// Mitsubishi GX Works2 project: EX2 (1) (1)   PLC: FX3G

// global labels: Global1
VAR_GLOBAL
  RM_Petel_Input AT D1100 : REAL;
  RG_Petel_Input AT D1100 : REAL;
  RG_Petel_Count AT D1200 : REAL;
  RG_Lemon_Input AT D1105 : REAL;
  RG_Lemon_Count AT D1205 : REAL;
  RG_Bear_Input AT D1110 : REAL;
  RG_Bear_Count AT D1215 : REAL;
  RG_Stables_Input AT D1120 : REAL;
  RG_Stables_Count AT D1220 : REAL;
END_VAR
VAR_GLOBAL CONSTANT
  Min_Petel_Amout : REAL := 385;
END_VAR
VAR_GLOBAL
  M2_Have_Petel AT M2 : BOOL;
END_VAR
VAR_GLOBAL CONSTANT
  Min_Petel_Amount : REAL := 105;
END_VAR
VAR_GLOBAL
  M3_Have_Lemon AT M3 : BOOL;
END_VAR
VAR_GLOBAL CONSTANT
  Min_Lemon_Amount : REAL := 665;
  Min_Bear_Amount : REAL := 70;
END_VAR
VAR_GLOBAL
  M4_Have_Bear AT M4 : BOOL;
END_VAR
VAR_GLOBAL CONSTANT
  Min_Stables_Amount : REAL := 210;
END_VAR
VAR_GLOBAL
  M5_Have_Stables AT M5 : BOOL;
  RG_Sample_Type_Value AT D1500 : REAL;
END_VAR
VAR_GLOBAL CONSTANT
  Con400 : INT := K400;
  Cons400 : REAL := 400;
END_VAR
VAR_GLOBAL
  M9_select_type AT M9 : BOOL;
END_VAR
VAR_GLOBAL CONSTANT
  Cons5 : REAL := 5;
END_VAR
VAR_GLOBAL
  TS5_end_making AT TS5 : BOOL;
  M91_regular AT M91 : BOOL;
END_VAR
VAR_GLOBAL CONSTANT
  Cons6 : REAL := 6;
  Cons10 : INT := 10;
END_VAR
VAR_GLOBAL
  TS6_end_making AT TS6 : BOOL;
  M92_pinok AT M92 : BOOL;
END_VAR
VAR_GLOBAL CONSTANT
  Petel_Amount : REAL := 280;
END_VAR
VAR_GLOBAL
  RG_Petel_Making AT D1400 : REAL;
END_VAR
VAR_GLOBAL CONSTANT
  Lemon_Amount_Petel : REAL := 35;
  Lemon_Amount_Lemon : REAL := 420;
END_VAR
VAR_GLOBAL
  RG_Lemon_Making AT D1410 : REAL;
END_VAR
VAR_GLOBAL CONSTANT
  Stables_Amount_Petel : REAL := 35;
  Steables_Amount_Lemon : REAL := 70;
  Petel_Amount_pinok : REAL := 385;
  Lemon_Amount_Petel_Pinok : REAL := 105;
  Lemon_Amount_Lemon_Pinok : REAL := 560;
  Stables_Amount_Petel_Pinok : REAL := 70;
  Steables_Amount_Lemon_Pinok : REAL := 140;
  Lemon_Amount_total : REAL := 455;
  Stables_Amount_total : REAL := 105;
  Lemon_Amount_total_pinok : REAL := 665;
  Stables_Amount_total_pinok : REAL := 210;
  Count5 : REAL := 5;
  Cons50 : WORD := 50;
  Cons0 : REAL;
END_VAR
VAR_GLOBAL
  RG_type_analog_value AT D1610 : REAL;
  X6Test AT X006 : BOOL;
  RG_Petel_Cooling AT D1404 : REAL;
  RG_Lemon_Cooling AT D1414 : REAL;
  TC7_cooling AT TC7 : BOOL;
END_VAR
VAR_GLOBAL CONSTANT
  Cons80 : WORD := 80;
END_VAR
VAR_GLOBAL
  M11_cooling AT M11 : BOOL;
  TS7_end_cooling AT TS7 : BOOL;
  Y4_TEST AT Y004 : BOOL;
END_VAR
VAR_GLOBAL CONSTANT
  Regular_Bear : REAL := 28;
END_VAR
VAR_GLOBAL
  RG_Mix_Regular AT D1450 : REAL;
END_VAR
VAR_GLOBAL CONSTANT
  Pinok_Bear : REAL := 70;
END_VAR
VAR_GLOBAL
  RG_Mix_Pinok AT D1460 : REAL;
  TC8_Mixing_Regular AT TC8 : BOOL;
END_VAR
VAR_GLOBAL CONSTANT
  Cons30 : WORD := 30;
END_VAR
VAR_GLOBAL
  TC9_Mixing_Pinok AT TC9 : BOOL;
  M10_Mixing AT M10 : BOOL;
  TS8_End_Mixing_Regual AT TS8 : BOOL;
  M0_Mix_Blinking AT M0 : BOOL;
  TS0_Output_Timer AT TS0 : BOOL;
  M20_Mix_Blinking_Help1 AT M20 : BOOL;
  TC0_Blinking1_Timer AT TC0 : BOOL;
  TC1_Blinking2_Timer AT TC1 : BOOL;
  TS1_Output_Timer2 AT TS1 : BOOL;
  M21_Mix_Blinking_Help2 AT M21 : BOOL;
  TS9_End_Mixing_Pinok AT TS9 : BOOL;
END_VAR
VAR_GLOBAL CONSTANT
  Const10 : REAL := 10;
END_VAR
VAR_GLOBAL
  X4_Packing AT X004 : BOOL;
  X0_packing_1_ice_cream AT X000 : BOOL;
  Y4_Work_ON_packing AT Y004 : BOOL;
END_VAR
VAR_GLOBAL CONSTANT
  Cons7 : WORD := 7;
END_VAR
VAR_GLOBAL
  RG_Ice_Output AT D1600 : REAL;
  RG_Packed_Ice_Cream AT D1700 : REAL;
END_VAR
VAR_GLOBAL CONSTANT
  Con1 : REAL := 1;
  Cons40 : REAL := 40;
END_VAR
VAR_GLOBAL
  RG_Packed_Ice_Cream_float AT D1710 : REAL;
  Y7_Working_day AT Y007 : BOOL;
  X5_Emergency AT X005 : BOOL;
  M7_End_Of_Day AT M7 : BOOL;
  X7_Start_Day AT X007 : BOOL;
  X1_Sample_Type AT X001 : BOOL;
  Y0_making AT Y000 : BOOL;
  X2_Cooling AT X002 : BOOL;
  Y2_Cooling AT Y002 : BOOL;
  X3_Temp AT X003 : BOOL;
  TC5_making AT TC5 : BOOL;
  TC6_making AT TC6 : BOOL;
  M15_packing AT M15 : BOOL;
  Y5_Mixing AT Y005 : BOOL;
  Y6_Mixing AT Y006 : BOOL;
  CS1_Packing_Finish AT CS1 : BOOL;
  CC1_Packing AT CC1 : BOOL;
  M12_end_cooling AT M12 : BOOL;
  M16_End_Packing AT M16 : BOOL;
  M17_packing_help AT M17 : BOOL;
  RG_analog2_Output AT D8282 : INT;
  RG_Sample_Type AT D8280 : INT;
END_VAR

// task Task_01 (event TRUE, interval 0, priority 31): POU_01

PROGRAM POU_01
(* structured ladder/FBD written out as ST: instructions are called as NAME(EN, inputs, outputs); _pN, _eN, _tN stand for wires *)
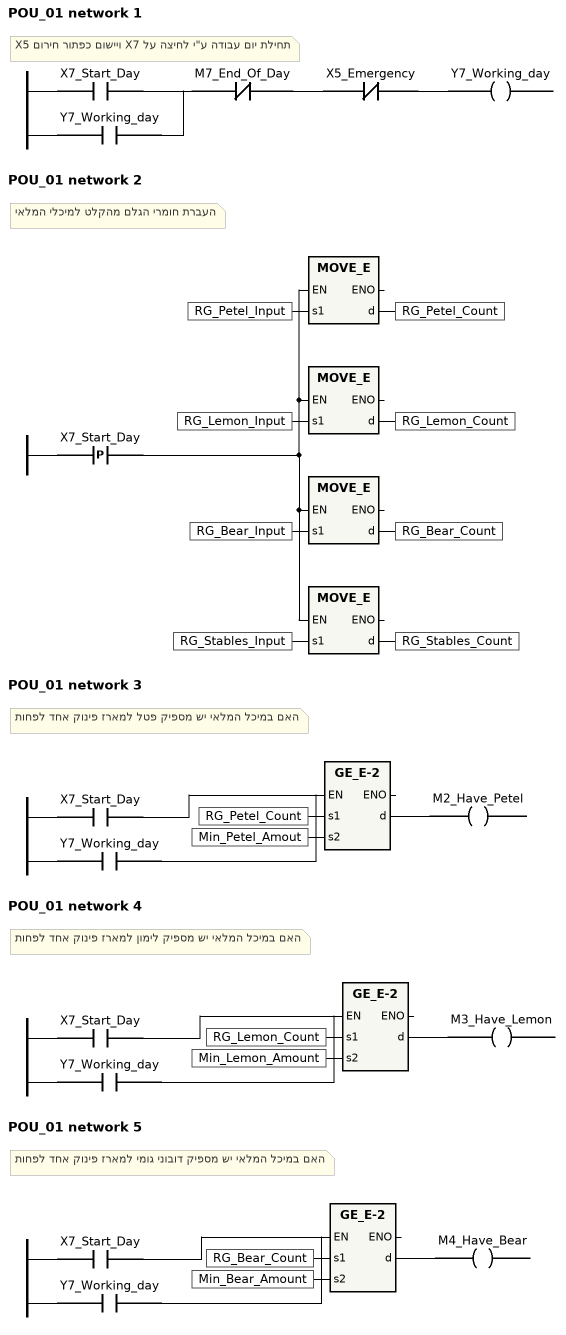
(* network 1 *)
(* תחילת יום עבודה ע"י לחיצה על X7 ויישום כפתור חירום X5 *)
Y7_Working_day := ((X7_Start_Day OR Y7_Working_day) AND NOT M7_End_Of_Day) AND NOT X5_Emergency;
(* network 2 *)
(* העברת חומרי הגלם מהקלט למיכלי המלאי *)
_p1 := LDP(TRUE, X7_Start_Day);
MOVE_E(_p1, RG_Petel_Input, RG_Petel_Count);
MOVE_E(_p1, RG_Lemon_Input, RG_Lemon_Count);
MOVE_E(_p1, RG_Bear_Input, RG_Bear_Count);
MOVE_E(_p1, RG_Stables_Input, RG_Stables_Count);
(* network 3 *)
(* האם במיכל המלאי יש מספיק פטל למארז פינוק אחד לפחות *)
GE_E(X7_Start_Day OR Y7_Working_day, RG_Petel_Count, Min_Petel_Amout, _t1);
M2_Have_Petel := _t1;
(* network 4 *)
(* האם במיכל המלאי יש מספיק לימון למארז פינוק אחד לפחות *)
GE_E(X7_Start_Day OR Y7_Working_day, RG_Lemon_Count, Min_Lemon_Amount, _t1);
M3_Have_Lemon := _t1;
(* network 5 *)
(* האם במיכל המלאי יש מספיק דובוני גומי למארז פינוק אחד לפחות *)
GE_E(X7_Start_Day OR Y7_Working_day, RG_Bear_Count, Min_Bear_Amount, _t1);
M4_Have_Bear := _t1;
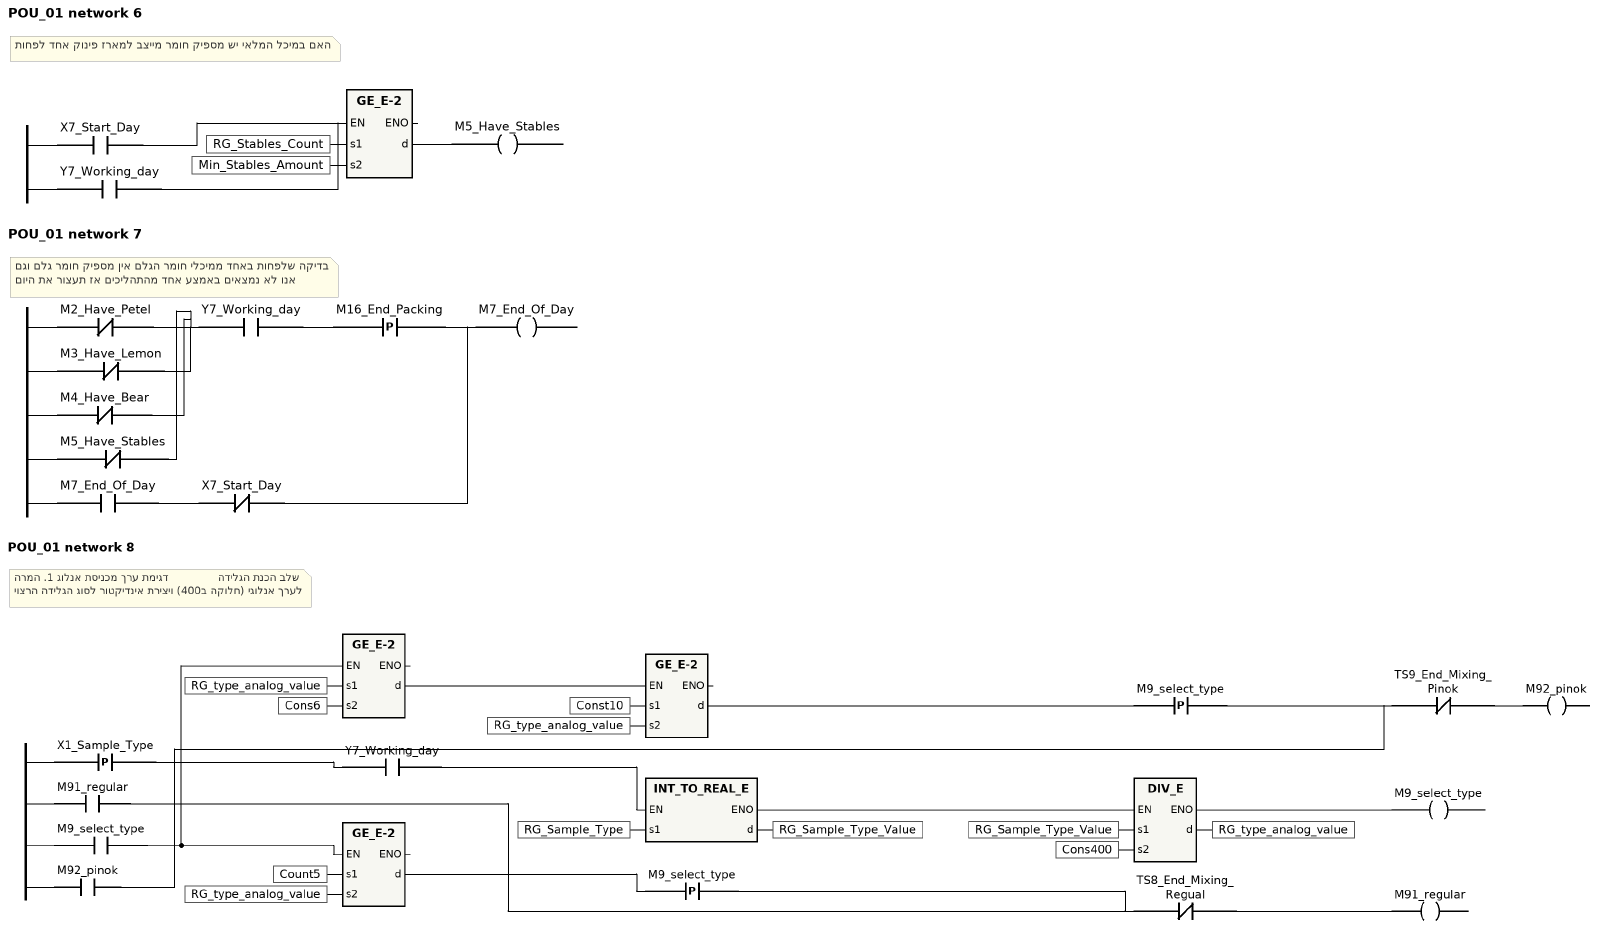
(* network 6 *)
(* האם במיכל המלאי יש מספיק חומר מייצב למארז פינוק אחד לפחות *)
GE_E(X7_Start_Day OR Y7_Working_day, RG_Stables_Count, Min_Stables_Amount, _t1);
M5_Have_Stables := _t1;
(* network 7 *)
(* בדיקה שלפחות באחד ממיכלי חומר הגלם אין מספיק חומר גלם וגם אנו לא נמצאים באמצע אחד מהתהליכים אז תעצור את היום *)
M7_End_Of_Day := ((((NOT M2_Have_Petel) OR (NOT M3_Have_Lemon) OR (NOT M4_Have_Bear) OR (NOT M5_Have_Stables)) AND Y7_Working_day) AND LDP(TRUE, M16_End_Packing)) OR (M7_End_Of_Day AND NOT X7_Start_Day);
(* network 8 *)
(* שלב הכנת הגלידה               דגימת ערך מכניסת אנלוג 1. המרה לערך אנלוגי (חלוקה ב400) ויצירת אינדיקטור לסוג הגלידה הרצוי *)
_e1 := INT_TO_REAL_E(LDP(TRUE, X1_Sample_Type) AND Y7_Working_day, RG_Sample_Type, RG_Sample_Type_Value);
_e2 := DIV_E(_e1, RG_Sample_Type_Value, Cons400, RG_type_analog_value);
M9_select_type := _e2;
GE_E(M9_select_type, Count5, RG_type_analog_value, _t3);
M91_regular := (M91_regular OR (_t3 AND LDP(TRUE, M9_select_type))) AND NOT TS8_End_Mixing_Regual;
GE_E(M9_select_type, RG_type_analog_value, Cons6, _t4);
GE_E(_t4, Const10, RG_type_analog_value, _t5);
M92_pinok := ((_t5 AND LDP(TRUE, M9_select_type)) OR M92_pinok) AND NOT TS9_End_Mixing_Pinok;
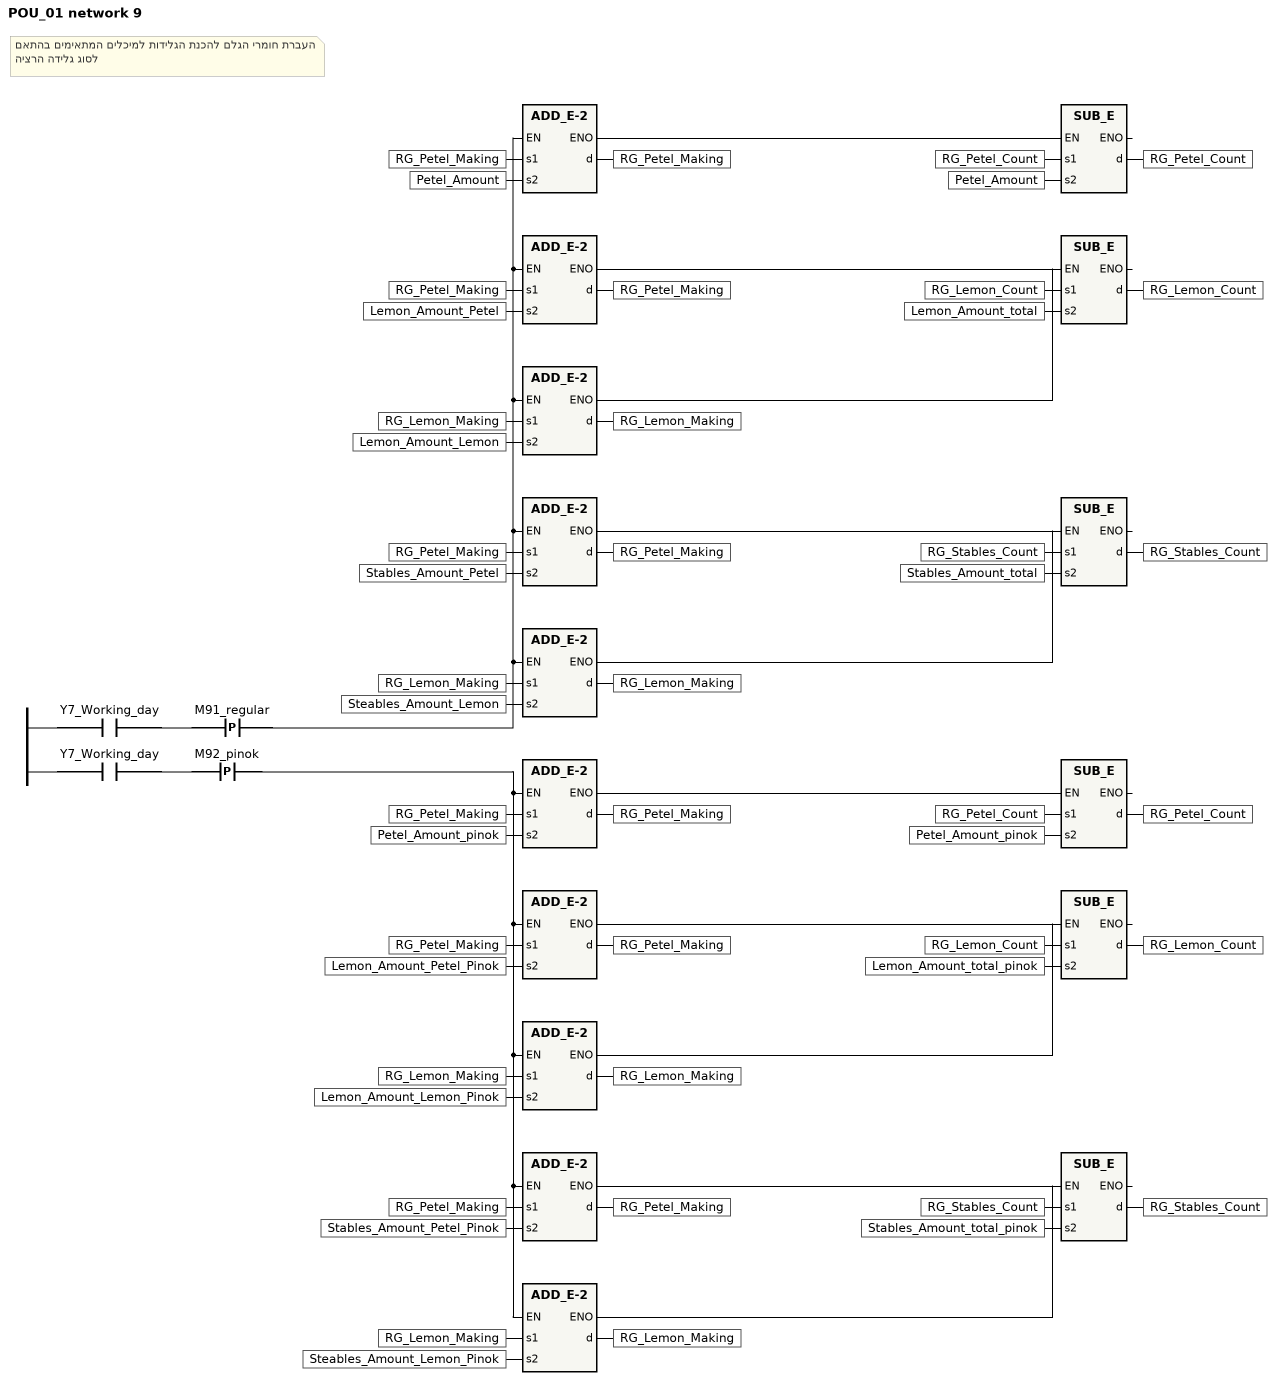
(* network 9 *)
(* העברת חומרי הגלם להכנת הגלידות למיכלים המתאימים בהתאם לסוג גלידה הרציה *)
_p1 := Y7_Working_day AND LDP(TRUE, M91_regular);
_e2 := ADD_E(_p1, RG_Petel_Making, Petel_Amount, RG_Petel_Making);
SUB_E(_e2, RG_Petel_Count, Petel_Amount, RG_Petel_Count);
_e3 := ADD_E(_p1, RG_Petel_Making, Lemon_Amount_Petel, RG_Petel_Making);
_e4 := ADD_E(_p1, RG_Lemon_Making, Lemon_Amount_Lemon, RG_Lemon_Making);
SUB_E(_e3 OR _e4, RG_Lemon_Count, Lemon_Amount_total, RG_Lemon_Count);
_e5 := ADD_E(_p1, RG_Petel_Making, Stables_Amount_Petel, RG_Petel_Making);
_e6 := ADD_E(_p1, RG_Lemon_Making, Steables_Amount_Lemon, RG_Lemon_Making);
SUB_E(_e5 OR _e6, RG_Stables_Count, Stables_Amount_total, RG_Stables_Count);
_p7 := Y7_Working_day AND LDP(TRUE, M92_pinok);
_e8 := ADD_E(_p7, RG_Petel_Making, Petel_Amount_pinok, RG_Petel_Making);
SUB_E(_e8, RG_Petel_Count, Petel_Amount_pinok, RG_Petel_Count);
_e9 := ADD_E(_p7, RG_Petel_Making, Lemon_Amount_Petel_Pinok, RG_Petel_Making);
_e10 := ADD_E(_p7, RG_Lemon_Making, Lemon_Amount_Lemon_Pinok, RG_Lemon_Making);
SUB_E(_e9 OR _e10, RG_Lemon_Count, Lemon_Amount_total_pinok, RG_Lemon_Count);
_e11 := ADD_E(_p7, RG_Petel_Making, Stables_Amount_Petel_Pinok, RG_Petel_Making);
_e12 := ADD_E(_p7, RG_Lemon_Making, Steables_Amount_Lemon_Pinok, RG_Lemon_Making);
SUB_E(_e11 OR _e12, RG_Stables_Count, Stables_Amount_total_pinok, RG_Stables_Count);
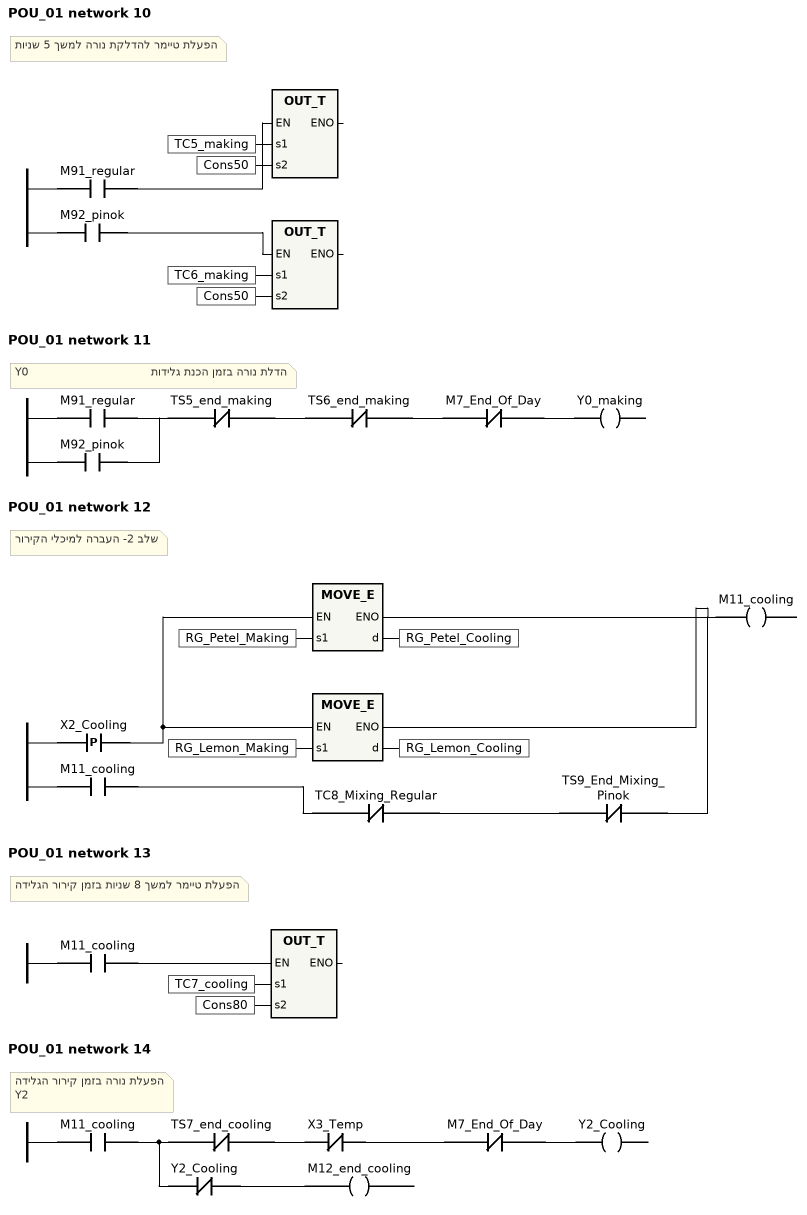
(* network 10 *)
(* הפעלת טיימר להדלקת נורה למשך 5 שניות *)
OUT_T(M91_regular, TC5_making, Cons50);
OUT_T(M92_pinok, TC6_making, Cons50);
(* network 11 *)
(* הדלת נורה בזמן הכנת גלידות                                   Y0 *)
Y0_making := (((M91_regular OR M92_pinok) AND NOT TS5_end_making) AND NOT TS6_end_making) AND NOT M7_End_Of_Day;
(* network 12 *)
(* שלב 2- העברה למיכלי הקירור *)
_p1 := LDP(TRUE, X2_Cooling);
_e2 := MOVE_E(_p1, RG_Petel_Making, RG_Petel_Cooling);
_e3 := MOVE_E(_p1, RG_Lemon_Making, RG_Lemon_Cooling);
M11_cooling := _e2 OR _e3 OR (M11_cooling AND NOT TC8_Mixing_Regular AND NOT TS9_End_Mixing_Pinok);
(* network 13 *)
(* הפעלת טיימר למשך 8 שניות בזמן קירור הגלידה *)
OUT_T(M11_cooling, TC7_cooling, Cons80);
(* network 14 *)
(* הפעלת נורה בזמן קירור הגלידה  / Y2 *)
Y2_Cooling := M11_cooling AND NOT TS7_end_cooling AND NOT X3_Temp AND NOT M7_End_Of_Day;
M12_end_cooling := M11_cooling AND NOT Y2_Cooling;
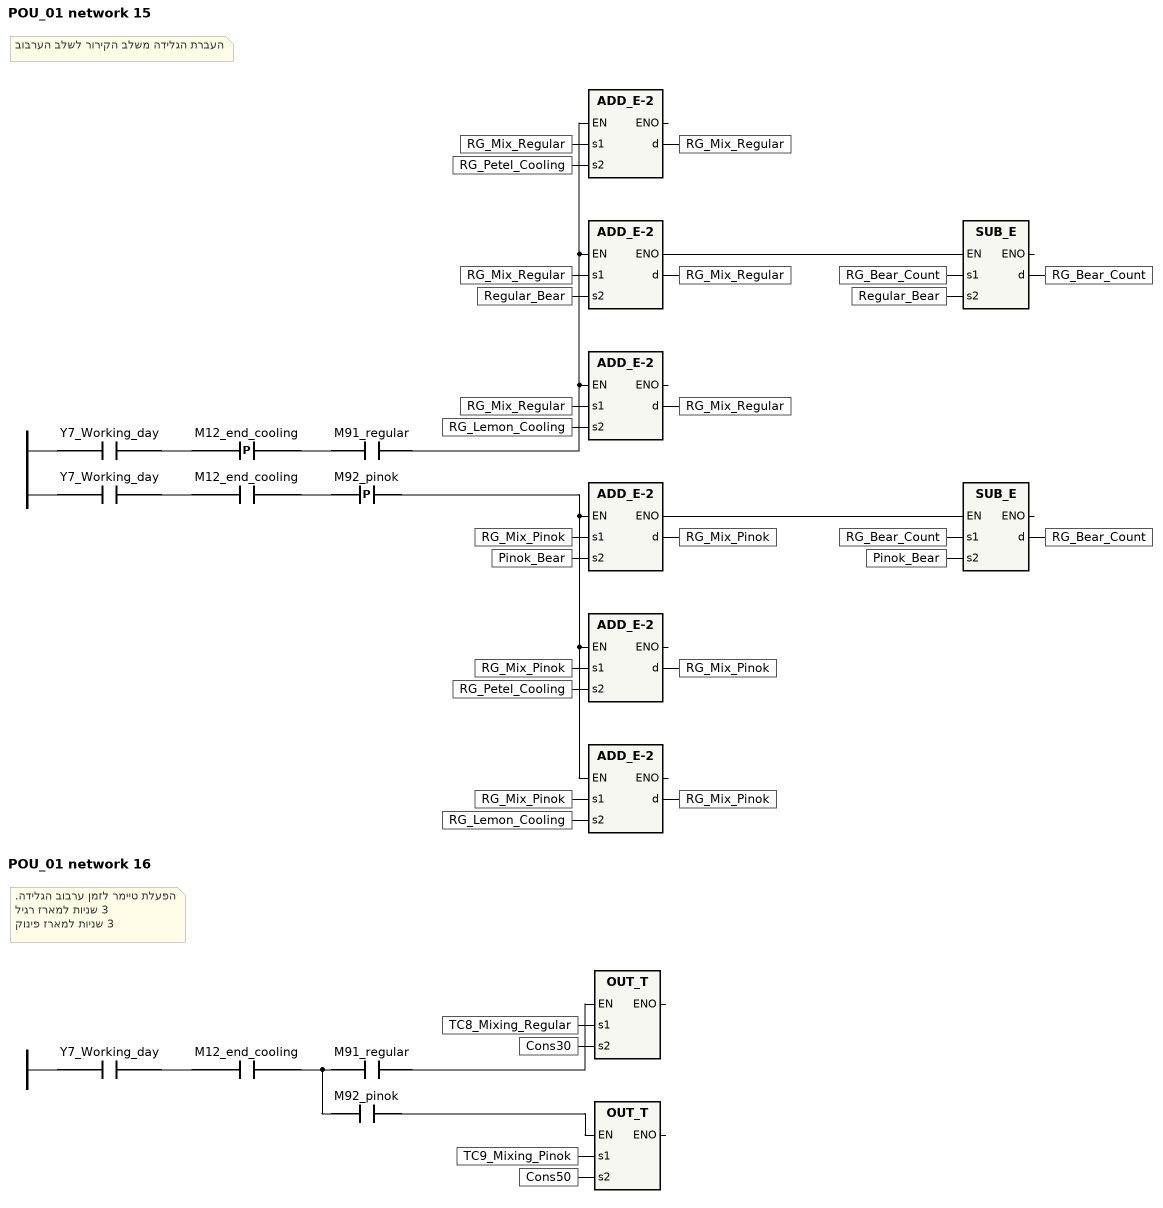
(* network 15 *)
(* העברת הגלידה משלב הקירור לשלב הערבוב *)
_p1 := Y7_Working_day AND LDP(TRUE, M12_end_cooling) AND M91_regular;
ADD_E(_p1, RG_Mix_Regular, RG_Petel_Cooling, RG_Mix_Regular);
ADD_E(_p1, RG_Mix_Regular, RG_Lemon_Cooling, RG_Mix_Regular);
_e2 := ADD_E(_p1, RG_Mix_Regular, Regular_Bear, RG_Mix_Regular);
SUB_E(_e2, RG_Bear_Count, Regular_Bear, RG_Bear_Count);
_p3 := Y7_Working_day AND M12_end_cooling AND LDP(TRUE, M92_pinok);
ADD_E(_p3, RG_Mix_Pinok, RG_Petel_Cooling, RG_Mix_Pinok);
ADD_E(_p3, RG_Mix_Pinok, RG_Lemon_Cooling, RG_Mix_Pinok);
_e4 := ADD_E(_p3, RG_Mix_Pinok, Pinok_Bear, RG_Mix_Pinok);
SUB_E(_e4, RG_Bear_Count, Pinok_Bear, RG_Bear_Count);
(* network 16 *)
(* הפעלת טיימר לזמן ערבוב הגלידה. / 3 שניות למארז רגיל / 3 שניות למארז פינוק *)
_p1 := Y7_Working_day AND M12_end_cooling;
OUT_T(_p1 AND M91_regular, TC8_Mixing_Regular, Cons30);
OUT_T(_p1 AND M92_pinok, TC9_Mixing_Pinok, Cons50);
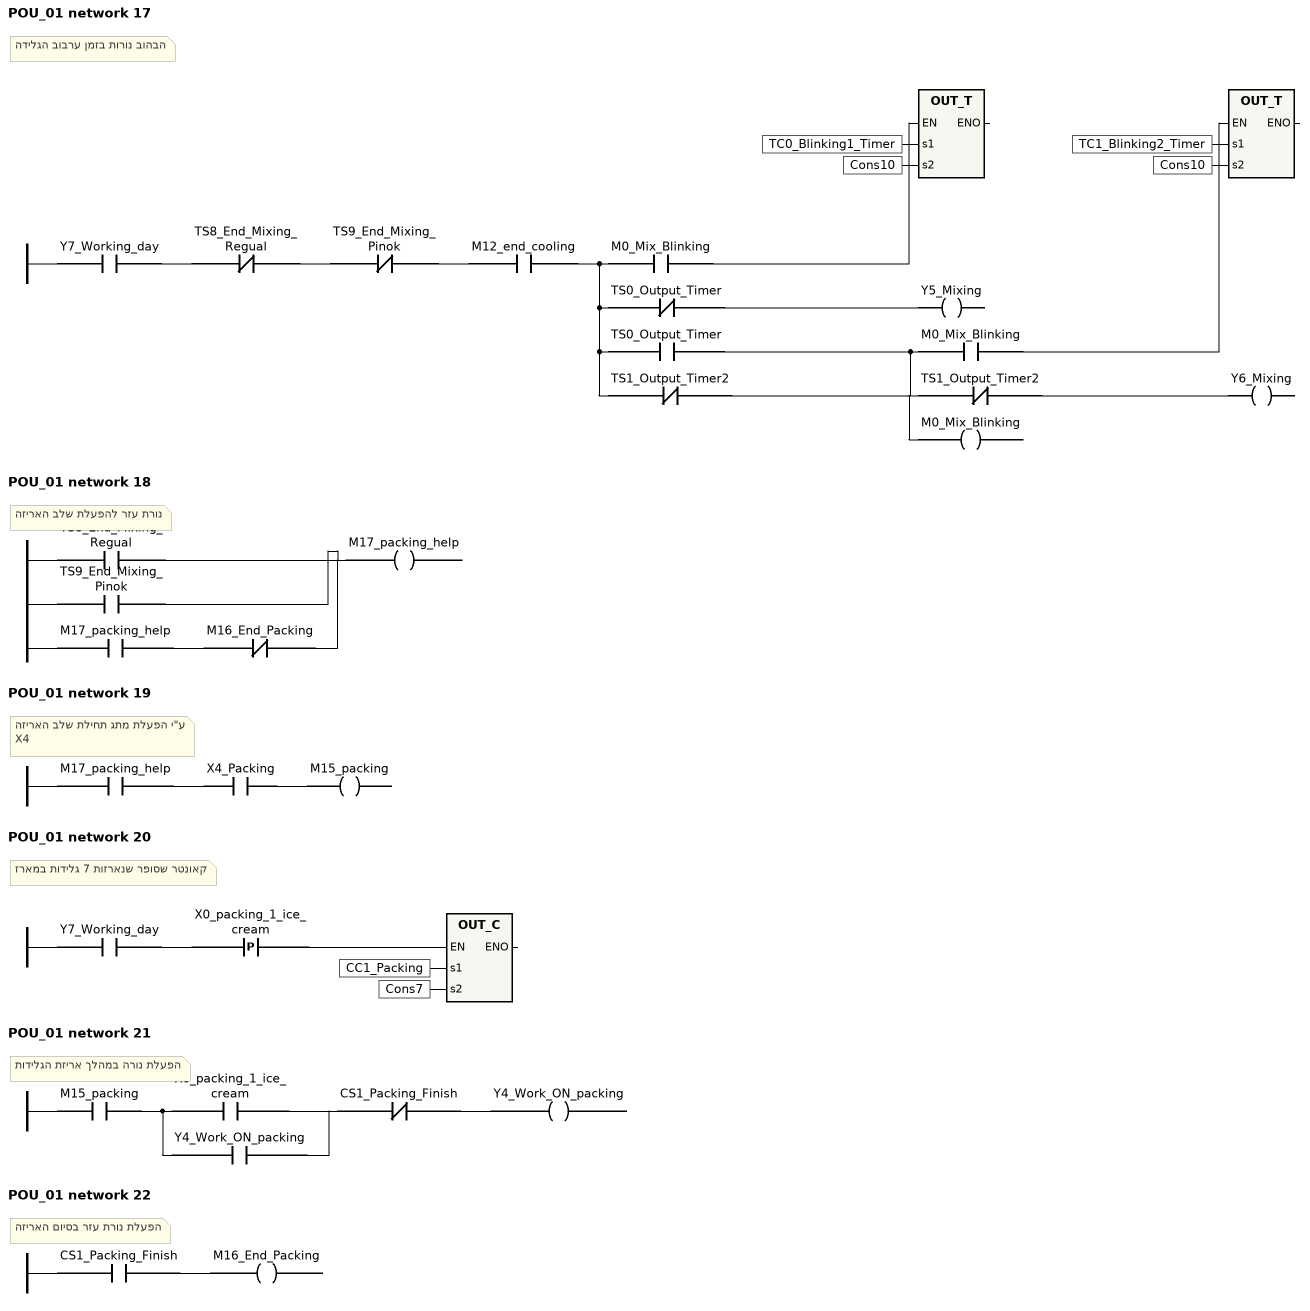
(* network 17 *)
(* הבהוב נורות בזמן ערבוב הגלידה *)
_p1 := Y7_Working_day AND NOT TS8_End_Mixing_Regual AND NOT TS9_End_Mixing_Pinok AND M12_end_cooling;
OUT_T(_p1 AND M0_Mix_Blinking, TC0_Blinking1_Timer, Cons10);
Y5_Mixing := _p1 AND NOT TS0_Output_Timer;
_p2 := _p1 AND TS0_Output_Timer;
OUT_T(_p2 AND M0_Mix_Blinking, TC1_Blinking2_Timer, Cons10);
Y6_Mixing := _p2 AND NOT TS1_Output_Timer2;
M0_Mix_Blinking := _p1 AND NOT TS1_Output_Timer2;
(* network 18 *)
(* נורת עזר להפעלת שלב האריזה *)
M17_packing_help := TS8_End_Mixing_Regual OR TS9_End_Mixing_Pinok OR (M17_packing_help AND NOT M16_End_Packing);
(* network 19 *)
(* ע"י הפעלת מתג תחילת שלב האריזה  / X4 *)
M15_packing := M17_packing_help AND X4_Packing;
(* network 20 *)
(* קאונטר שסופר שנארזות 7 גלידות במארז *)
OUT_C(Y7_Working_day AND LDP(TRUE, X0_packing_1_ice_cream), CC1_Packing, Cons7);
(* network 21 *)
(* הפעלת נורה במהלך אריזת הגלידות *)
Y4_Work_ON_packing := ((M15_packing AND X0_packing_1_ice_cream) OR (M15_packing AND Y4_Work_ON_packing)) AND NOT CS1_Packing_Finish;
(* network 22 *)
(* הפעלת נורת עזר בסיום האריזה *)
M16_End_Packing := CS1_Packing_Finish;
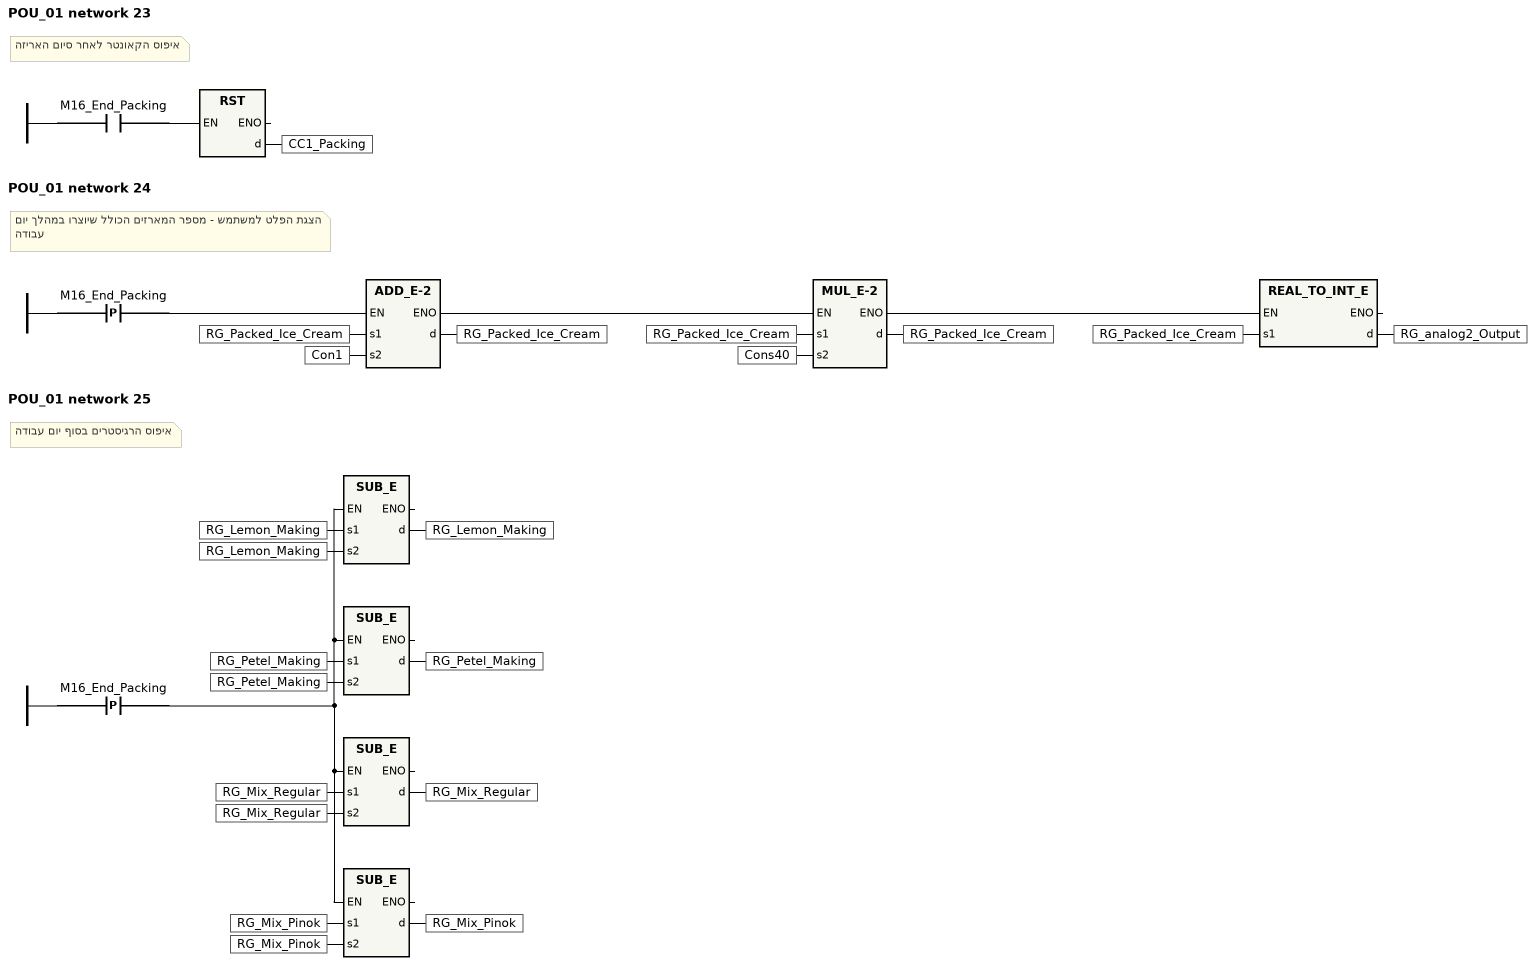
(* network 23 *)
(* איפוס הקאונטר לאחר סיום האריזה *)
RST(M16_End_Packing, CC1_Packing);
(* network 24 *)
(* הצגת הפלט למשתמש - מספר המארזים הכולל שיוצרו במהלך יום עבודה *)
_e1 := ADD_E(LDP(TRUE, M16_End_Packing), RG_Packed_Ice_Cream, Con1, RG_Packed_Ice_Cream);
_e2 := MUL_E(_e1, RG_Packed_Ice_Cream, Cons40, RG_Packed_Ice_Cream);
REAL_TO_INT_E(_e2, RG_Packed_Ice_Cream, RG_analog2_Output);
(* network 25 *)
(* איפוס הרגיסטרים בסוף יום עבודה *)
_p1 := LDP(TRUE, M16_End_Packing);
SUB_E(_p1, RG_Lemon_Making, RG_Lemon_Making, RG_Lemon_Making);
SUB_E(_p1, RG_Petel_Making, RG_Petel_Making, RG_Petel_Making);
SUB_E(_p1, RG_Mix_Regular, RG_Mix_Regular, RG_Mix_Regular);
SUB_E(_p1, RG_Mix_Pinok, RG_Mix_Pinok, RG_Mix_Pinok);
END_PROGRAM
